INTERFACE ITask

PROPERTY Done : BOOL
GET
END_GET
END_PROPERTY

END_INTERFACE

(* stored: Version 1.1.0.1, ProductVersion 3.1.4024.5
   Itf ITask: Id {12f0ee69-8b2e-45a9-8407-04acf1a7e096}
   Property Done: Id {75d26d18-3e85-4883-bef6-c3e9611690cb}
   Get Get: Id {dfebaec5-8940-4c3a-81d7-c329021bada1} *)
